PROGRAM MAIN
VAR
	fbAxisEthMaster: FB_AxisEthMaster;
	M1: FB_AxisMaster;
	M2: FB_AxisMaster;
	M3: FB_AxisMaster;
	bFirstCycle: BOOL := TRUE;
END_VAR

// Set the initial configs
IF bFirstCycle THEN
	M2.stConfigSet.ref_vel := 10;
	M2.stConfigSet.max_vel := 20;
	M2.stConfigSet.man_fast := 15;
	M2.stConfigSet.man_slow := 5;
	M2.stConfigSet.enc_scale := 0.001;
	M2.stConfigSet.max_current := 1100;
	M3.stConfigSet.ref_vel := 11;
	M3.stConfigSet.max_vel := 21;
	M3.stConfigSet.man_fast := 16;
	M3.stConfigSet.man_slow := 6;
	M3.stConfigSet.enc_scale := 0.002;
	M3.stConfigSet.max_current := 1234;
	bFirstCycle := FALSE;
END_IF

// Bring MASTER to OP once SLAVEs are PRE-OP
fbAxisEthMaster(bExecute:=M1.bInitPreOp AND M2.bInitPreOp AND M3.bInitPreOp);

// Enable and pass Cfg
M1(bEnable:=TRUE,
	bInitCfg:=FALSE,
	bCfgRO:=FALSE,
	bUseLimits:=FALSE);
M2(bEnable:=TRUE,
	bInitCfg:=TRUE,
	bCfgRO:=FALSE,
	nEncCh:=1);
M3(bEnable:=TRUE,
	bInitCfg:=TRUE,
	bCfgRO:=TRUE,
	nEncCh:=2);

END_PROGRAM

(* stored: Version 1.1.0.1, ProductVersion 3.1.4020.12
   POU MAIN: Id {372593b4-1746-4f2d-8630-4bf2374df086}, SpecialFunc None *)
